FUNCTION_BLOCK VAV_CTL (* Variable Air Volume Controller *)
  (* Standard: 61499-1; ApplicationDomain: HVAC; Function: Control; Type: VAV; Description: Variable Air Volume Controller *)
  (* Version 0.0, 2006-04-27, JHC, Holobloc Inc *)
  (* Compiler header: package fb.rt.hvac; *)
  (* Compiler Java Sun JDK 1.5.0 *)
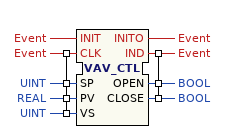
  EVENT_INPUT
    INIT; (* Initialization Request *)
    CLK WITH SP, PV, VS; (* Periodic Execution Clock *)
  END_EVENT
  EVENT_OUTPUT
    INITO; (* Initialization Confirm *)
    IND WITH OPEN, CLOSE; (* OPEN/CLOSE command value change *)
  END_EVENT
  VAR_INPUT
    SP : UINT := 50; (* Set point, deg F *)
    PV : REAL := 70.0; (* Zone Temperature, deg F *)
    VS : UINT; (* Velocity Sensor Reading *)
  END_VAR
  VAR_OUTPUT
    OPEN : BOOL; (* Damper OPEN command *)
    CLOSE : BOOL; (* Damper CLOSE command *)
  END_VAR
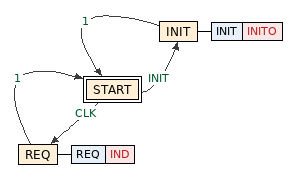
  EC_STATES
    START; (* Initial State *)
    INIT : INIT -> INITO; (* Initialization *)
    REQ : REQ -> IND; (* Normal execution *)
  END_STATES
  EC_TRANSITIONS
    START TO INIT := INIT;
    INIT TO START := 1;
    START TO REQ := CLK;
    REQ TO START := 1;
  END_TRANSITIONS
  ALGORITHM INIT IN ST: (* Initialization algorithm *)

  END_ALGORITHM
  ALGORITHM REQ IN ST: (* Normally executed algorithm *)

  END_ALGORITHM
END_FUNCTION_BLOCK
